// TIA Portal V17 export
// export: Created 2025-03-10T12:18:45.1065076Z, ExportSetting WithDefaults, DisplayName Totally Integrated Automation Portal, DisplayVersion V17 Update 8, DisplayName TIA Portal Openness, DisplayVersion V17 Update 8, DisplayName TIA Portal Version Control Interface, DisplayVersion V17, DisplayName SINAMICS Startdrive Advanced, DisplayVersion V17 SP2, DisplayName SINAMICS Startdrive G110M, G120, G120C, G120D, G120P, G115D, DisplayVersion V17 SP2, DisplayName SINAMICS Startdrive G130, G150, S120, S150, SINAMICS MV, S210, DisplayVersion V17 SP2, DisplayName STEP 7 Professional, DisplayVersion V17 Update 8, DisplayName SINUMERIK ONE STEP 7 Toolbox, DisplayVersion V17 Update 12, DisplayName SINUMERIK 840D sl STEP 7 Toolbox, DisplayVersion V17 Update 12, DisplayName STEP 7 Safety, DisplayVersion V17 Update 6, DisplayName WinCC Advanced, DisplayVersion V17 Update 8
FUNCTION_BLOCK "FB21011_POWDER_FEEDER_GENERAL"   // FB21011, LAD
TITLE = FB21011 POWDER FEEDER GENERAL
{ S7_Optimized_Access := 'TRUE' }
VERSION : 0.1
// stored: AutoNumber false, IsIECCheckEnabled false, IsRetainMemResEnabled false, MemoryReserve 100, SetENOAutomatically false, UDAEnableTagReadback false
   VAR_INPUT
      iPOWDER_FEEDER_BRAKER_FAULT : Bool;
      iOPERATION_MODE_LINE_1 : Word;
      iOPERATION_MODE_LINE_2 : Word;
      iOPERATION_MODE_MATCHED_LINE_1 : Bool;
      iOPERATION_MODE_MATCHED_LINE_2 : Bool;
      iFEEDER_STATE_LINE_1 : Word;
      iFEEDER_STATE_LINE_2 : Word;
      iCARRIERGAS_STATUS_LINE_1 : Bool;
      iCARRIERGAS_STATUS_LINE_2 : Bool;
      iENABLED : Bool;
   END_VAR
   VAR_OUTPUT
      oCONNECT_POWDER_FEEDER : Bool;
      oOPERATION_MODE : Word;
      oPRODUCTION_MODE : Word;
      oSYSTEM_MODE : Word;
      oSTATION_IS_ALARMS : Bool;
      oSwitchoncondition_on : Bool;
      oSwitchoncondition_off : Bool;
      oMotion_Active_Right : Bool;
      oMotion_Active_Left : Bool;
      oLimit_right : Bool;
      oLimit_left : Bool;
      oALARM_MISMATCH_FAULT : Bool;
      oALARM_FEEDER_PROFINET_MODE_FAULT : Bool;
   END_VAR
   VAR
      DATA : "POWDER FEEDER GENERAL";
      INPUT_SETTINGS : Struct
         UNIT_NUMBER : Int;
         FEEDER_NUMBER : Int;
      END_STRUCT;
   END_VAR
   VAR_TEMP
      OPTIONS_OFF : Bool;
      OPTIONS_ON : Bool;
      HOPPER_1 : Bool;
      HOPPER_2 : Bool;
      DB_NUMBER : DInt;
   END_VAR
   VAR_TEMP   // added for the SCL form of the ladder/FBD networks
      _w1 : Bool;
   END_VAR
BEGIN

NETWORK
TITLE = READ INSTANCE DB NUMBER
      L     DINO;
      +     10#800000;
      T     #DB_NUMBER;

REGION Network 2: OPTIONS OFF / Options Off
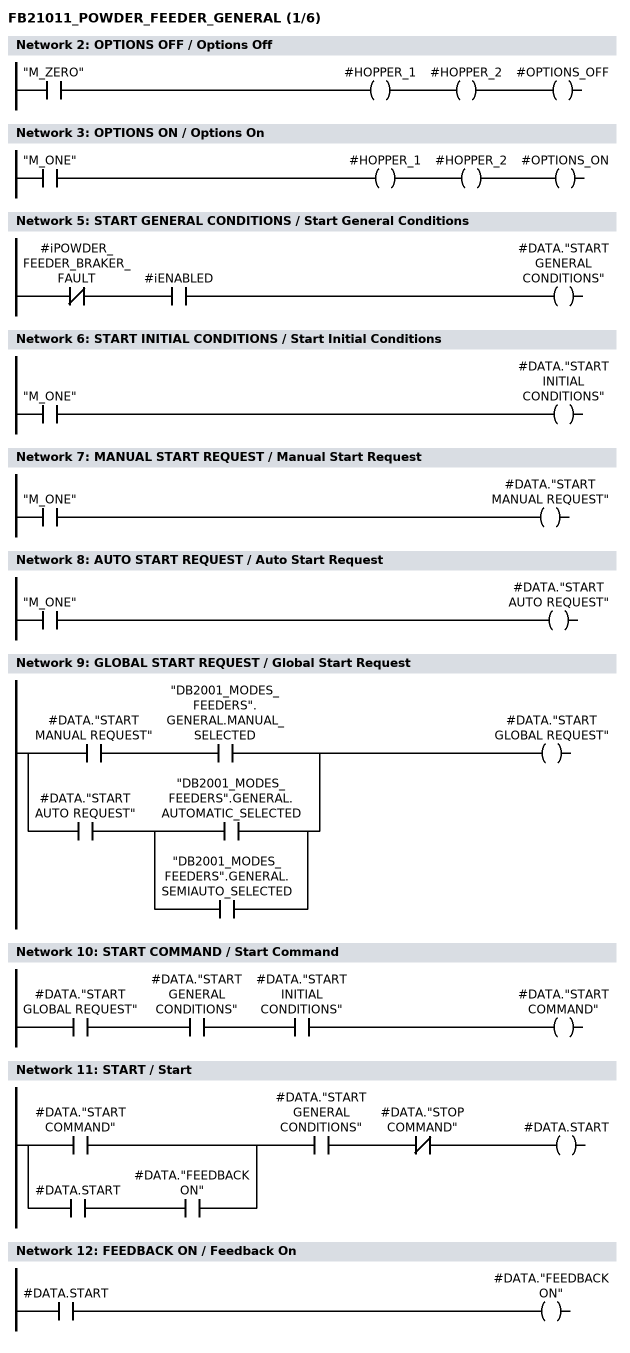
   RUNG wire#powerrail
      Contact( "M_ZERO" )
      Coil( #HOPPER_1 )
      Coil( #HOPPER_2 )
      Coil( #OPTIONS_OFF )
   END_RUNG
   // the same network as SCL:
   #HOPPER_1 := "M_ZERO";
   #HOPPER_2 := "M_ZERO";
   #OPTIONS_OFF := "M_ZERO";
END_REGION

REGION Network 3: OPTIONS ON / Options On
   RUNG wire#powerrail
      Contact( "M_ONE" )
      Coil( #HOPPER_1 )
      Coil( #HOPPER_2 )
      Coil( #OPTIONS_ON )
   END_RUNG
   // the same network as SCL:
   #HOPPER_1 := "M_ONE";
   #HOPPER_2 := "M_ONE";
   #OPTIONS_ON := "M_ONE";
END_REGION

REGION Network 4: INPUT / Input
END_REGION

REGION Network 5: START GENERAL CONDITIONS / Start General Conditions
   RUNG wire#powerrail
      I_Contact( #iPOWDER_FEEDER_BRAKER_FAULT )
      Contact( #iENABLED )
      Coil( #DATA."START GENERAL CONDITIONS" )
   END_RUNG
   // the same network as SCL:
   #DATA."START GENERAL CONDITIONS" := NOT #iPOWDER_FEEDER_BRAKER_FAULT AND #iENABLED;
END_REGION

REGION Network 6: START INITIAL CONDITIONS / Start Initial Conditions
   RUNG wire#powerrail
      Contact( "M_ONE" )
      Coil( #DATA."START INITIAL CONDITIONS" )
   END_RUNG
   // the same network as SCL:
   #DATA."START INITIAL CONDITIONS" := "M_ONE";
END_REGION

REGION Network 7: MANUAL START REQUEST / Manual Start Request
   RUNG wire#powerrail
      Contact( "M_ONE" )
      Coil( #DATA."START MANUAL REQUEST" )
   END_RUNG
   // the same network as SCL:
   #DATA."START MANUAL REQUEST" := "M_ONE";
END_REGION

REGION Network 8: AUTO START REQUEST / Auto Start Request
   RUNG wire#powerrail
      Contact( "M_ONE" )
      Coil( #DATA."START AUTO REQUEST" )
   END_RUNG
   // the same network as SCL:
   #DATA."START AUTO REQUEST" := "M_ONE";
END_REGION

REGION Network 9: GLOBAL START REQUEST / Global Start Request
   RUNG wire#powerrail
      Contact( #DATA."START MANUAL REQUEST" )
      Contact( "DB2001_MODES_FEEDERS".GENERAL.MANUAL_SELECTED )
      wire#w1
      Coil( #DATA."START GLOBAL REQUEST" )
   END_RUNG
   RUNG wire#powerrail
      Contact( #DATA."START AUTO REQUEST" )
      wire#w2
      Contact( "DB2001_MODES_FEEDERS".GENERAL.AUTOMATIC_SELECTED )
   END_RUNG wire#w1
   RUNG wire#w2
      Contact( "DB2001_MODES_FEEDERS".GENERAL.SEMIAUTO_SELECTED )
   END_RUNG wire#w1
   // the same network as SCL:
   #DATA."START GLOBAL REQUEST" := (#DATA."START MANUAL REQUEST" AND "DB2001_MODES_FEEDERS".GENERAL.MANUAL_SELECTED) OR (#DATA."START AUTO REQUEST" AND ("DB2001_MODES_FEEDERS".GENERAL.AUTOMATIC_SELECTED OR "DB2001_MODES_FEEDERS".GENERAL.SEMIAUTO_SELECTED));
END_REGION

REGION Network 10: START COMMAND / Start Command
   RUNG wire#powerrail
      Contact( #DATA."START GLOBAL REQUEST" )
      Contact( #DATA."START GENERAL CONDITIONS" )
      Contact( #DATA."START INITIAL CONDITIONS" )
      Coil( #DATA."START COMMAND" )
   END_RUNG
   // the same network as SCL:
   #DATA."START COMMAND" := #DATA."START GLOBAL REQUEST" AND #DATA."START GENERAL CONDITIONS" AND #DATA."START INITIAL CONDITIONS";
END_REGION

REGION Network 11: START / Start
   RUNG wire#powerrail
      Contact( #DATA."START COMMAND" )
      wire#w1
      Contact( #DATA."START GENERAL CONDITIONS" )
      I_Contact( #DATA."STOP COMMAND" )
      Coil( #DATA.START )
   END_RUNG
   RUNG wire#powerrail
      Contact( #DATA.START )
      Contact( #DATA."FEEDBACK ON" )
   END_RUNG wire#w1
   // the same network as SCL:
   #DATA.START := (#DATA."START COMMAND" OR (#DATA.START AND #DATA."FEEDBACK ON")) AND #DATA."START GENERAL CONDITIONS" AND NOT #DATA."STOP COMMAND";
END_REGION

REGION Network 12: FEEDBACK ON / Feedback On
   RUNG wire#powerrail
      Contact( #DATA.START )
      Coil( #DATA."FEEDBACK ON" )
   END_RUNG
   // the same network as SCL:
   #DATA."FEEDBACK ON" := #DATA.START;
END_REGION

REGION Network 13: STOP GENERAL CONDITIONS / Stop General Conditions
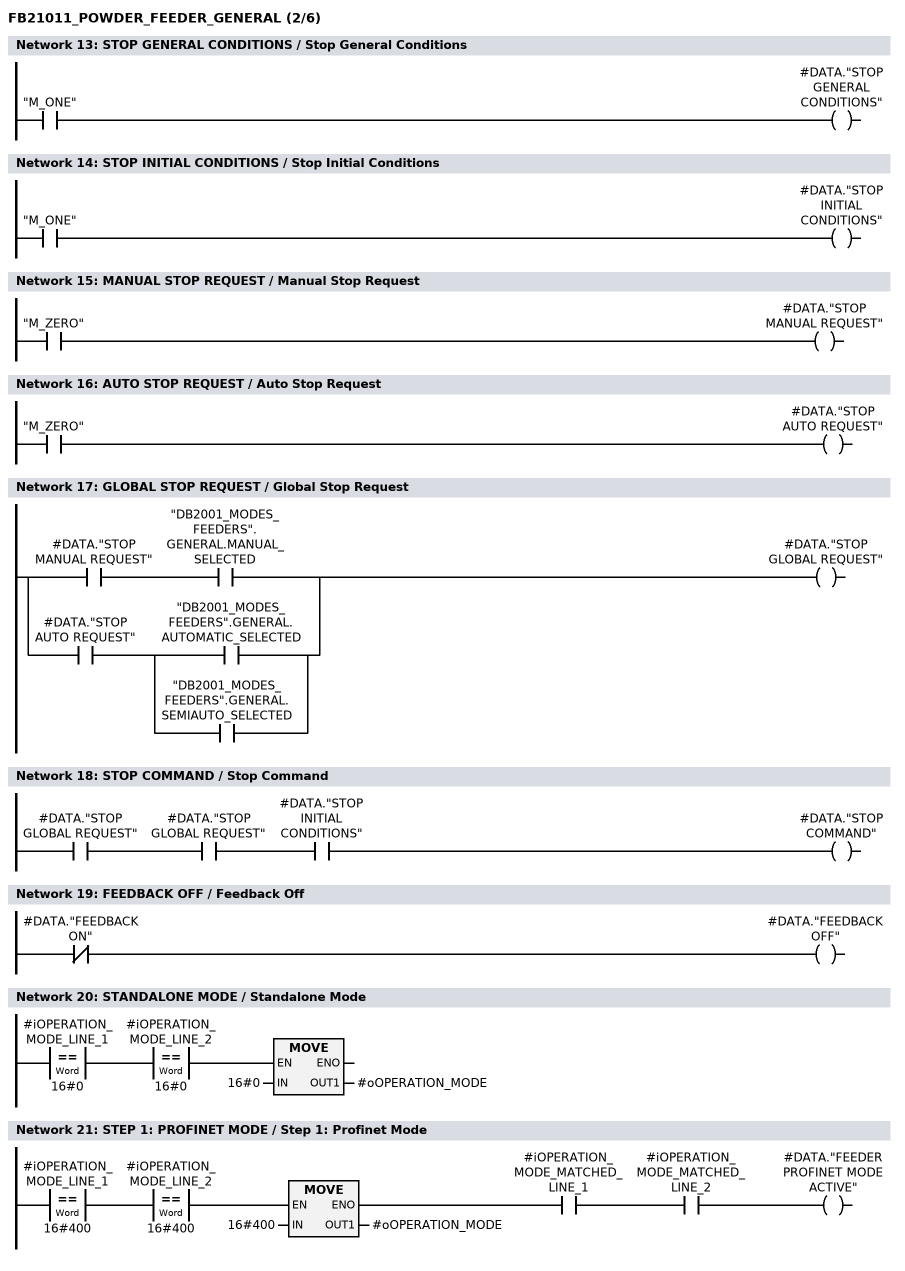
   RUNG wire#powerrail
      Contact( "M_ONE" )
      Coil( #DATA."STOP GENERAL CONDITIONS" )
   END_RUNG
   // the same network as SCL:
   #DATA."STOP GENERAL CONDITIONS" := "M_ONE";
END_REGION

REGION Network 14: STOP INITIAL CONDITIONS / Stop Initial Conditions
   RUNG wire#powerrail
      Contact( "M_ONE" )
      Coil( #DATA."STOP INITIAL CONDITIONS" )
   END_RUNG
   // the same network as SCL:
   #DATA."STOP INITIAL CONDITIONS" := "M_ONE";
END_REGION

REGION Network 15: MANUAL STOP REQUEST / Manual Stop Request
   RUNG wire#powerrail
      Contact( "M_ZERO" )
      Coil( #DATA."STOP MANUAL REQUEST" )
   END_RUNG
   // the same network as SCL:
   #DATA."STOP MANUAL REQUEST" := "M_ZERO";
END_REGION

REGION Network 16: AUTO STOP REQUEST / Auto Stop Request
   RUNG wire#powerrail
      Contact( "M_ZERO" )
      Coil( #DATA."STOP AUTO REQUEST" )
   END_RUNG
   // the same network as SCL:
   #DATA."STOP AUTO REQUEST" := "M_ZERO";
END_REGION

REGION Network 17: GLOBAL STOP REQUEST / Global Stop Request
   RUNG wire#powerrail
      Contact( #DATA."STOP MANUAL REQUEST" )
      Contact( "DB2001_MODES_FEEDERS".GENERAL.MANUAL_SELECTED )
      wire#w1
      Coil( #DATA."STOP GLOBAL REQUEST" )
   END_RUNG
   RUNG wire#powerrail
      Contact( #DATA."STOP AUTO REQUEST" )
      wire#w2
      Contact( "DB2001_MODES_FEEDERS".GENERAL.AUTOMATIC_SELECTED )
   END_RUNG wire#w1
   RUNG wire#w2
      Contact( "DB2001_MODES_FEEDERS".GENERAL.SEMIAUTO_SELECTED )
   END_RUNG wire#w1
   // the same network as SCL:
   #DATA."STOP GLOBAL REQUEST" := (#DATA."STOP MANUAL REQUEST" AND "DB2001_MODES_FEEDERS".GENERAL.MANUAL_SELECTED) OR (#DATA."STOP AUTO REQUEST" AND ("DB2001_MODES_FEEDERS".GENERAL.AUTOMATIC_SELECTED OR "DB2001_MODES_FEEDERS".GENERAL.SEMIAUTO_SELECTED));
END_REGION

REGION Network 18: STOP COMMAND / Stop Command
   RUNG wire#powerrail
      Contact( #DATA."STOP GLOBAL REQUEST" )
      Contact( #DATA."STOP GLOBAL REQUEST" )
      Contact( #DATA."STOP INITIAL CONDITIONS" )
      Coil( #DATA."STOP COMMAND" )
   END_RUNG
   // the same network as SCL:
   #DATA."STOP COMMAND" := #DATA."STOP GLOBAL REQUEST" AND #DATA."STOP GLOBAL REQUEST" AND #DATA."STOP INITIAL CONDITIONS";
END_REGION

REGION Network 19: FEEDBACK OFF / Feedback Off
   RUNG wire#powerrail
      I_Contact( #DATA."FEEDBACK ON" )
      Coil( #DATA."FEEDBACK OFF" )
   END_RUNG
   // the same network as SCL:
   #DATA."FEEDBACK OFF" := NOT #DATA."FEEDBACK ON";
END_REGION

REGION Network 20: STANDALONE MODE / Standalone Mode
   RUNG wire#powerrail
      { S7_Templates := "SrcType := Word" } EQ_Contact(in1 := #iOPERATION_MODE_LINE_1, in2 := 16#0)
      { S7_Templates := "SrcType := Word" } EQ_Contact(in1 := #iOPERATION_MODE_LINE_2, in2 := 16#0)
      Move(in := 16#0, out1 => #oOPERATION_MODE)
   END_RUNG
   // the same network as SCL:
   IF (#iOPERATION_MODE_LINE_1 = 16#0) AND (#iOPERATION_MODE_LINE_2 = 16#0) THEN
       #oOPERATION_MODE := 16#0;
   END_IF;
END_REGION

REGION Network 21: STEP 1: PROFINET MODE / Step 1: Profinet Mode
   RUNG wire#powerrail
      { S7_Templates := "SrcType := Word" } EQ_Contact(in1 := #iOPERATION_MODE_LINE_1, in2 := 16#400)
      { S7_Templates := "SrcType := Word" } EQ_Contact(in1 := #iOPERATION_MODE_LINE_2, in2 := 16#400)
      Move(in := 16#400, out1 => #oOPERATION_MODE)
      Contact( #iOPERATION_MODE_MATCHED_LINE_1 )
      Contact( #iOPERATION_MODE_MATCHED_LINE_2 )
      Coil( #DATA."FEEDER PROFINET MODE ACTIVE" )
   END_RUNG
   // the same network as SCL:
   #_w1 := (#iOPERATION_MODE_LINE_1 = 16#400) AND (#iOPERATION_MODE_LINE_2 = 16#400);
   IF #_w1 THEN #oOPERATION_MODE := 16#400; END_IF;
   #DATA."FEEDER PROFINET MODE ACTIVE" := #_w1 AND #iOPERATION_MODE_MATCHED_LINE_1 AND #iOPERATION_MODE_MATCHED_LINE_2;
END_REGION

REGION Network 22: STEP 2: PRODUCTION MODE / Step 2: Production Mode
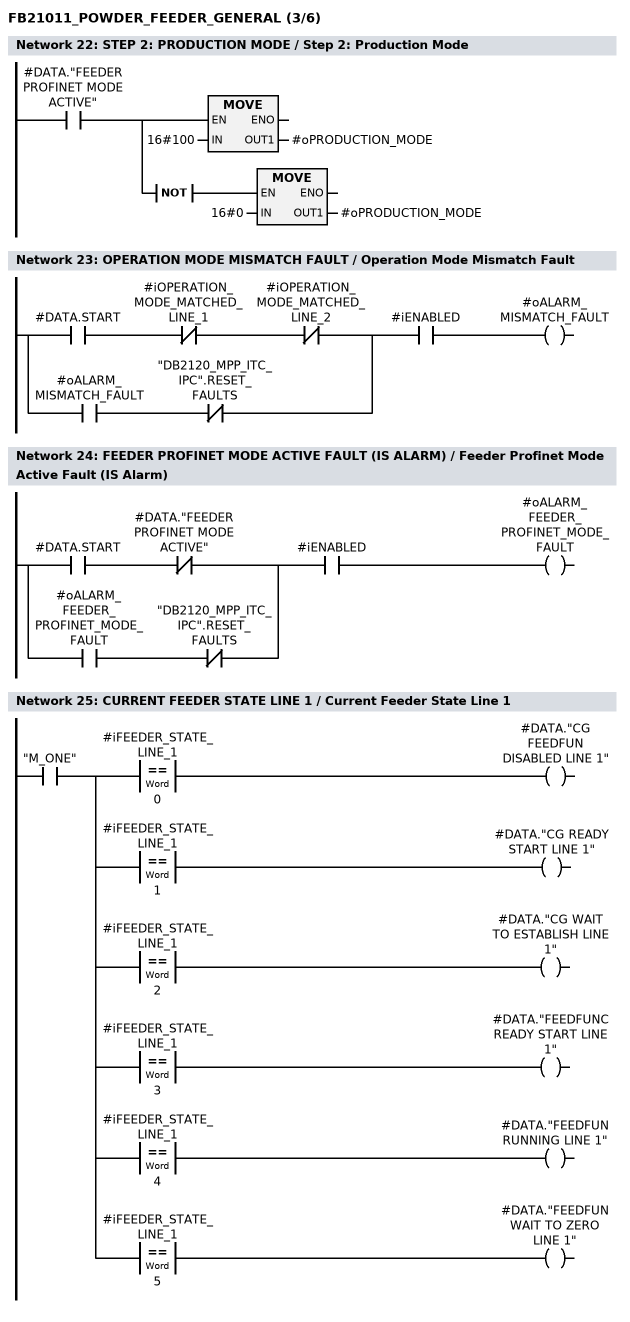
   RUNG wire#powerrail
      Contact( #DATA."FEEDER PROFINET MODE ACTIVE" )
      wire#w1
      Move(in := 16#100, out1 => #oPRODUCTION_MODE)
   END_RUNG
   RUNG wire#w1
      Not()
      Move(in := 16#0, out1 => #oPRODUCTION_MODE)
   END_RUNG
   // the same network as SCL:
   IF #DATA."FEEDER PROFINET MODE ACTIVE" THEN #oPRODUCTION_MODE := 16#100; END_IF;
   IF NOT #DATA."FEEDER PROFINET MODE ACTIVE" THEN #oPRODUCTION_MODE := 16#0; END_IF;
END_REGION

REGION Network 23: OPERATION MODE MISMATCH FAULT / Operation Mode Mismatch Fault
   RUNG wire#powerrail
      Contact( #DATA.START )
      I_Contact( #iOPERATION_MODE_MATCHED_LINE_1 )
      I_Contact( #iOPERATION_MODE_MATCHED_LINE_2 )
      wire#w1
      Contact( #iENABLED )
      Coil( #oALARM_MISMATCH_FAULT )
   END_RUNG
   RUNG wire#powerrail
      Contact( #oALARM_MISMATCH_FAULT )
      I_Contact( "DB2120_MPP_ITC_IPC".RESET_FAULTS )
   END_RUNG wire#w1
   // the same network as SCL:
   #oALARM_MISMATCH_FAULT := ((#DATA.START AND NOT #iOPERATION_MODE_MATCHED_LINE_1 AND NOT #iOPERATION_MODE_MATCHED_LINE_2) OR (#oALARM_MISMATCH_FAULT AND NOT "DB2120_MPP_ITC_IPC".RESET_FAULTS)) AND #iENABLED;
END_REGION

REGION Network 24: FEEDER PROFINET MODE ACTIVE FAULT (IS ALARM) / Feeder Profinet Mode Active Fault (IS Alarm)
   RUNG wire#powerrail
      Contact( #DATA.START )
      I_Contact( #DATA."FEEDER PROFINET MODE ACTIVE" )
      wire#w1
      Contact( #iENABLED )
      Coil( #oALARM_FEEDER_PROFINET_MODE_FAULT )
   END_RUNG
   RUNG wire#powerrail
      Contact( #oALARM_FEEDER_PROFINET_MODE_FAULT )
      I_Contact( "DB2120_MPP_ITC_IPC".RESET_FAULTS )
   END_RUNG wire#w1
   // the same network as SCL:
   #oALARM_FEEDER_PROFINET_MODE_FAULT := ((#DATA.START AND NOT #DATA."FEEDER PROFINET MODE ACTIVE") OR (#oALARM_FEEDER_PROFINET_MODE_FAULT AND NOT "DB2120_MPP_ITC_IPC".RESET_FAULTS)) AND #iENABLED;
END_REGION

REGION Network 25: CURRENT FEEDER STATE LINE 1 / Current Feeder State Line 1
   RUNG wire#powerrail
      Contact( "M_ONE" )
      wire#w1
      { S7_Templates := "SrcType := Word" } EQ_Contact(in1 := #iFEEDER_STATE_LINE_1, in2 := 0)
      Coil( #DATA."CG FEEDFUN DISABLED LINE 1" )
   END_RUNG
   RUNG wire#w1
      { S7_Templates := "SrcType := Word" } EQ_Contact(in1 := #iFEEDER_STATE_LINE_1, in2 := 1)
      Coil( #DATA."CG READY START LINE 1" )
   END_RUNG
   RUNG wire#w1
      { S7_Templates := "SrcType := Word" } EQ_Contact(in1 := #iFEEDER_STATE_LINE_1, in2 := 2)
      Coil( #DATA."CG WAIT TO ESTABLISH LINE 1" )
   END_RUNG
   RUNG wire#w1
      { S7_Templates := "SrcType := Word" } EQ_Contact(in1 := #iFEEDER_STATE_LINE_1, in2 := 3)
      Coil( #DATA."FEEDFUNC READY START LINE 1" )
   END_RUNG
   RUNG wire#w1
      { S7_Templates := "SrcType := Word" } EQ_Contact(in1 := #iFEEDER_STATE_LINE_1, in2 := 4)
      Coil( #DATA."FEEDFUN RUNNING LINE 1" )
   END_RUNG
   RUNG wire#w1
      { S7_Templates := "SrcType := Word" } EQ_Contact(in1 := #iFEEDER_STATE_LINE_1, in2 := 5)
      Coil( #DATA."FEEDFUN WAIT TO ZERO LINE 1" )
   END_RUNG
   // the same network as SCL:
   #DATA."CG FEEDFUN DISABLED LINE 1" := "M_ONE" AND (#iFEEDER_STATE_LINE_1 = 0);
   #DATA."CG READY START LINE 1" := "M_ONE" AND (#iFEEDER_STATE_LINE_1 = 1);
   #DATA."CG WAIT TO ESTABLISH LINE 1" := "M_ONE" AND (#iFEEDER_STATE_LINE_1 = 2);
   #DATA."FEEDFUNC READY START LINE 1" := "M_ONE" AND (#iFEEDER_STATE_LINE_1 = 3);
   #DATA."FEEDFUN RUNNING LINE 1" := "M_ONE" AND (#iFEEDER_STATE_LINE_1 = 4);
   #DATA."FEEDFUN WAIT TO ZERO LINE 1" := "M_ONE" AND (#iFEEDER_STATE_LINE_1 = 5);
END_REGION

REGION Network 26: CURRENT FEEDER STATE LINE 2 / Current Feeder State Line 2
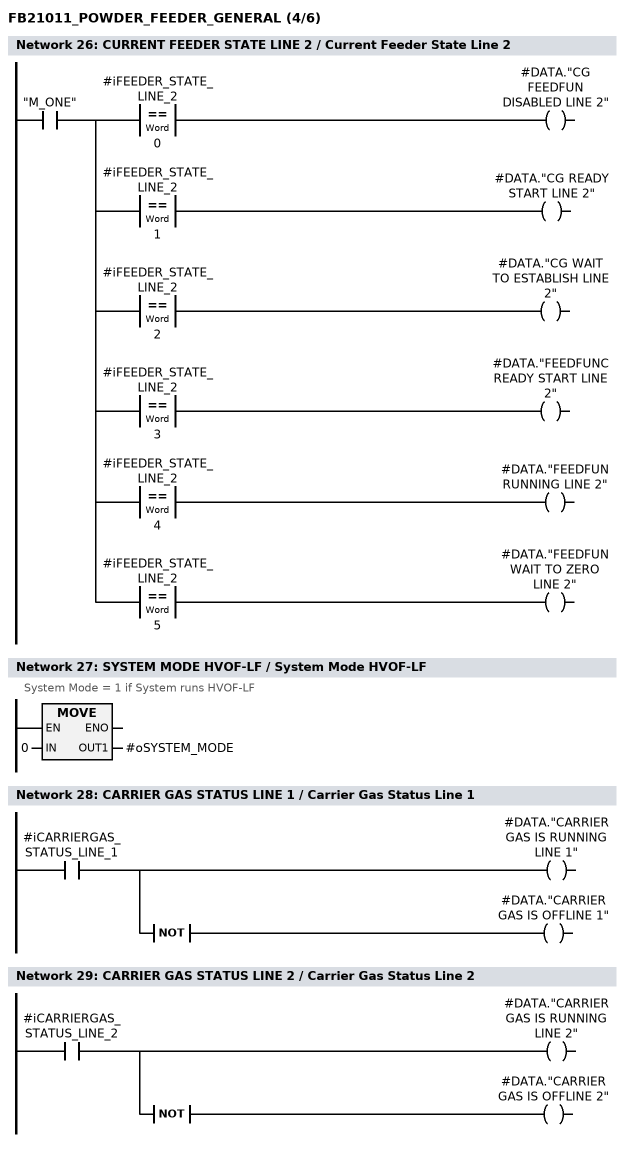
   RUNG wire#powerrail
      Contact( "M_ONE" )
      wire#w1
      { S7_Templates := "SrcType := Word" } EQ_Contact(in1 := #iFEEDER_STATE_LINE_2, in2 := 0)
      Coil( #DATA."CG FEEDFUN DISABLED LINE 2" )
   END_RUNG
   RUNG wire#w1
      { S7_Templates := "SrcType := Word" } EQ_Contact(in1 := #iFEEDER_STATE_LINE_2, in2 := 1)
      Coil( #DATA."CG READY START LINE 2" )
   END_RUNG
   RUNG wire#w1
      { S7_Templates := "SrcType := Word" } EQ_Contact(in1 := #iFEEDER_STATE_LINE_2, in2 := 2)
      Coil( #DATA."CG WAIT TO ESTABLISH LINE 2" )
   END_RUNG
   RUNG wire#w1
      { S7_Templates := "SrcType := Word" } EQ_Contact(in1 := #iFEEDER_STATE_LINE_2, in2 := 3)
      Coil( #DATA."FEEDFUNC READY START LINE 2" )
   END_RUNG
   RUNG wire#w1
      { S7_Templates := "SrcType := Word" } EQ_Contact(in1 := #iFEEDER_STATE_LINE_2, in2 := 4)
      Coil( #DATA."FEEDFUN RUNNING LINE 2" )
   END_RUNG
   RUNG wire#w1
      { S7_Templates := "SrcType := Word" } EQ_Contact(in1 := #iFEEDER_STATE_LINE_2, in2 := 5)
      Coil( #DATA."FEEDFUN WAIT TO ZERO LINE 2" )
   END_RUNG
   // the same network as SCL:
   #DATA."CG FEEDFUN DISABLED LINE 2" := "M_ONE" AND (#iFEEDER_STATE_LINE_2 = 0);
   #DATA."CG READY START LINE 2" := "M_ONE" AND (#iFEEDER_STATE_LINE_2 = 1);
   #DATA."CG WAIT TO ESTABLISH LINE 2" := "M_ONE" AND (#iFEEDER_STATE_LINE_2 = 2);
   #DATA."FEEDFUNC READY START LINE 2" := "M_ONE" AND (#iFEEDER_STATE_LINE_2 = 3);
   #DATA."FEEDFUN RUNNING LINE 2" := "M_ONE" AND (#iFEEDER_STATE_LINE_2 = 4);
   #DATA."FEEDFUN WAIT TO ZERO LINE 2" := "M_ONE" AND (#iFEEDER_STATE_LINE_2 = 5);
END_REGION

REGION Network 27: SYSTEM MODE HVOF-LF / System Mode HVOF-LF
   // System Mode = 1 if System runs HVOF-LF
   RUNG wire#powerrail
      Move(in := 0, out1 => #oSYSTEM_MODE)
   END_RUNG
   // the same network as SCL:
   #oSYSTEM_MODE := 0;
END_REGION

REGION Network 28: CARRIER GAS STATUS LINE 1 / Carrier Gas Status Line 1
   RUNG wire#powerrail
      Contact( #iCARRIERGAS_STATUS_LINE_1 )
      wire#w1
      Coil( #DATA."CARRIER GAS IS RUNNING LINE 1" )
   END_RUNG
   RUNG wire#w1
      Not()
      Coil( #DATA."CARRIER GAS IS OFFLINE 1" )
   END_RUNG
   // the same network as SCL:
   #DATA."CARRIER GAS IS RUNNING LINE 1" := #iCARRIERGAS_STATUS_LINE_1;
   #DATA."CARRIER GAS IS OFFLINE 1" := NOT #iCARRIERGAS_STATUS_LINE_1;
END_REGION

REGION Network 29: CARRIER GAS STATUS LINE 2 / Carrier Gas Status Line 2
   RUNG wire#powerrail
      Contact( #iCARRIERGAS_STATUS_LINE_2 )
      wire#w1
      Coil( #DATA."CARRIER GAS IS RUNNING LINE 2" )
   END_RUNG
   RUNG wire#w1
      Not()
      Coil( #DATA."CARRIER GAS IS OFFLINE 2" )
   END_RUNG
   // the same network as SCL:
   #DATA."CARRIER GAS IS RUNNING LINE 2" := #iCARRIERGAS_STATUS_LINE_2;
   #DATA."CARRIER GAS IS OFFLINE 2" := NOT #iCARRIERGAS_STATUS_LINE_2;
END_REGION

REGION Network 30: INMEDIATE STOP ALARMS / Inmediate Stop Alarms
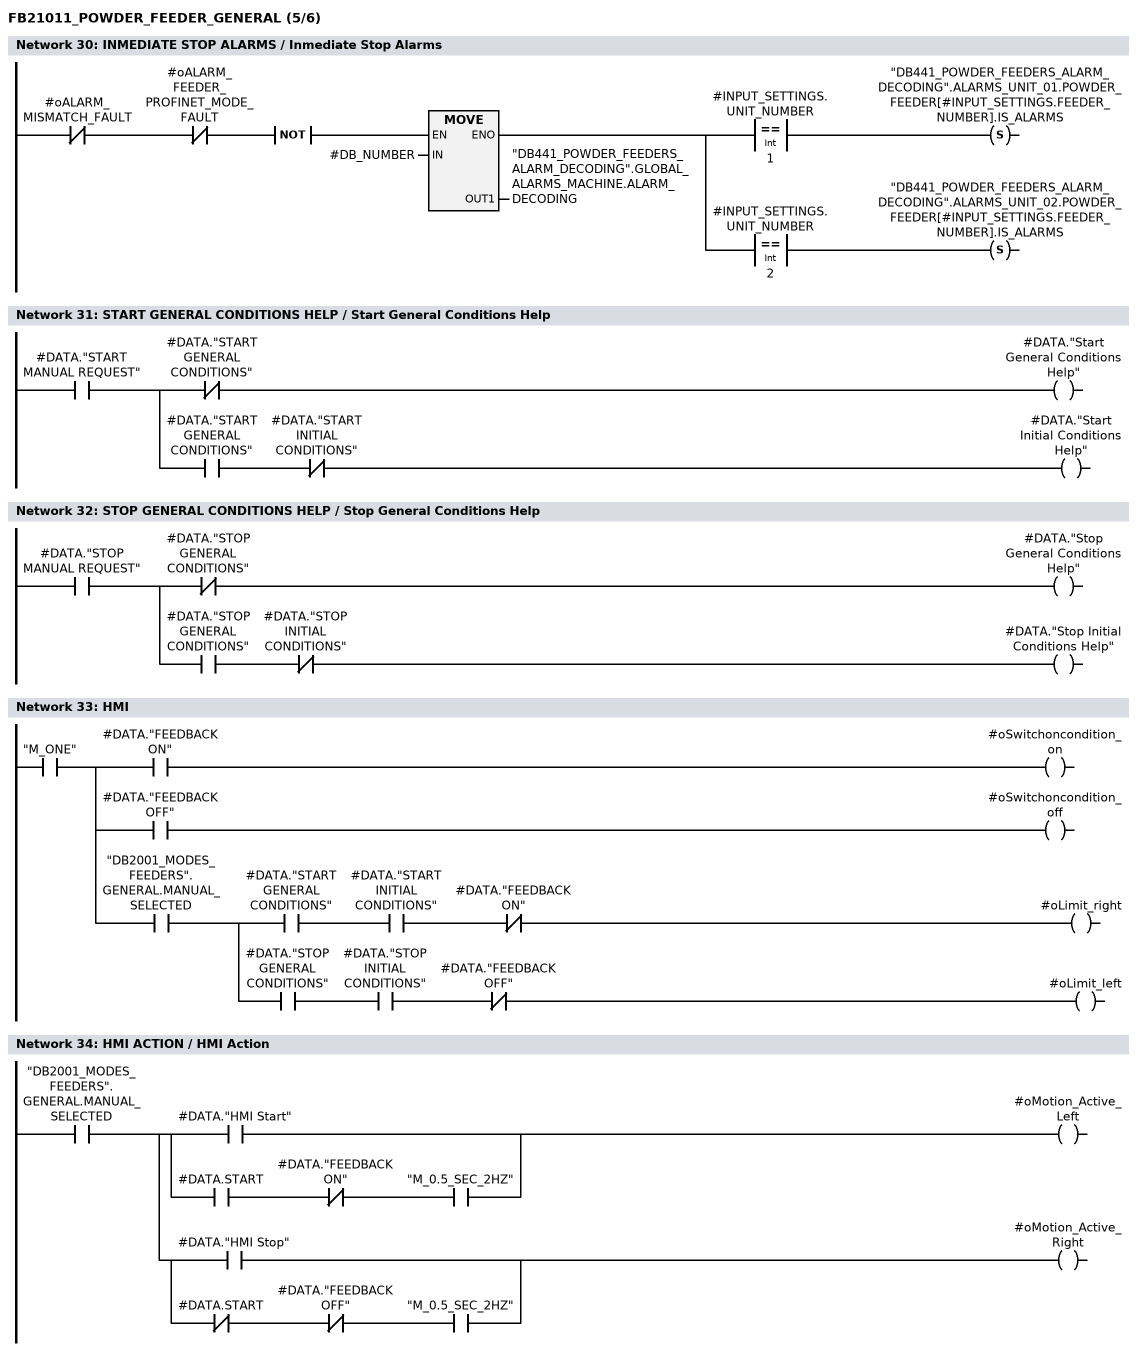
   RUNG wire#powerrail
      I_Contact( #oALARM_MISMATCH_FAULT )
      I_Contact( #oALARM_FEEDER_PROFINET_MODE_FAULT )
      Not()
      Move(in := #DB_NUMBER, out1 => "DB441_POWDER_FEEDERS_ALARM_DECODING".GLOBAL_ALARMS_MACHINE.ALARM_DECODING)
      wire#w1
      { S7_Templates := "SrcType := Int" } EQ_Contact(in1 := #INPUT_SETTINGS.UNIT_NUMBER, in2 := 1)
      S_Coil( "DB441_POWDER_FEEDERS_ALARM_DECODING".ALARMS_UNIT_01.POWDER_FEEDER[#INPUT_SETTINGS.FEEDER_NUMBER].IS_ALARMS )
   END_RUNG
   RUNG wire#w1
      { S7_Templates := "SrcType := Int" } EQ_Contact(in1 := #INPUT_SETTINGS.UNIT_NUMBER, in2 := 2)
      S_Coil( "DB441_POWDER_FEEDERS_ALARM_DECODING".ALARMS_UNIT_02.POWDER_FEEDER[#INPUT_SETTINGS.FEEDER_NUMBER].IS_ALARMS )
   END_RUNG
   // the same network as SCL:
   #_w1 := NOT (NOT #oALARM_MISMATCH_FAULT AND NOT #oALARM_FEEDER_PROFINET_MODE_FAULT);
   IF #_w1 THEN
       "DB441_POWDER_FEEDERS_ALARM_DECODING".GLOBAL_ALARMS_MACHINE.ALARM_DECODING := #DB_NUMBER;
   END_IF;
   IF #_w1 AND (#INPUT_SETTINGS.UNIT_NUMBER = 1) THEN
       "DB441_POWDER_FEEDERS_ALARM_DECODING".ALARMS_UNIT_01.POWDER_FEEDER[#INPUT_SETTINGS.FEEDER_NUMBER].IS_ALARMS := TRUE;
   END_IF;
   IF #_w1 AND (#INPUT_SETTINGS.UNIT_NUMBER = 2) THEN
       "DB441_POWDER_FEEDERS_ALARM_DECODING".ALARMS_UNIT_02.POWDER_FEEDER[#INPUT_SETTINGS.FEEDER_NUMBER].IS_ALARMS := TRUE;
   END_IF;
END_REGION

REGION Network 31: START GENERAL CONDITIONS HELP / Start General Conditions Help
   RUNG wire#powerrail
      Contact( #DATA."START MANUAL REQUEST" )
      wire#w1
      I_Contact( #DATA."START GENERAL CONDITIONS" )
      Coil( #DATA."Start General Conditions Help" )
   END_RUNG
   RUNG wire#w1
      Contact( #DATA."START GENERAL CONDITIONS" )
      I_Contact( #DATA."START INITIAL CONDITIONS" )
      Coil( #DATA."Start Initial Conditions Help" )
   END_RUNG
   // the same network as SCL:
   #DATA."Start General Conditions Help" := #DATA."START MANUAL REQUEST" AND NOT #DATA."START GENERAL CONDITIONS";
   #DATA."Start Initial Conditions Help" := #DATA."START MANUAL REQUEST" AND #DATA."START GENERAL CONDITIONS" AND NOT #DATA."START INITIAL CONDITIONS";
END_REGION

REGION Network 32: STOP GENERAL CONDITIONS HELP / Stop General Conditions Help
   RUNG wire#powerrail
      Contact( #DATA."STOP MANUAL REQUEST" )
      wire#w1
      I_Contact( #DATA."STOP GENERAL CONDITIONS" )
      Coil( #DATA."Stop General Conditions Help" )
   END_RUNG
   RUNG wire#w1
      Contact( #DATA."STOP GENERAL CONDITIONS" )
      I_Contact( #DATA."STOP INITIAL CONDITIONS" )
      Coil( #DATA."Stop Initial Conditions Help" )
   END_RUNG
   // the same network as SCL:
   #DATA."Stop General Conditions Help" := #DATA."STOP MANUAL REQUEST" AND NOT #DATA."STOP GENERAL CONDITIONS";
   #DATA."Stop Initial Conditions Help" := #DATA."STOP MANUAL REQUEST" AND #DATA."STOP GENERAL CONDITIONS" AND NOT #DATA."STOP INITIAL CONDITIONS";
END_REGION

REGION Network 33: HMI
   RUNG wire#powerrail
      Contact( "M_ONE" )
      wire#w1
      Contact( #DATA."FEEDBACK ON" )
      Coil( #oSwitchoncondition_on )
   END_RUNG
   RUNG wire#w1
      Contact( #DATA."FEEDBACK OFF" )
      Coil( #oSwitchoncondition_off )
   END_RUNG
   RUNG wire#w1
      Contact( "DB2001_MODES_FEEDERS".GENERAL.MANUAL_SELECTED )
      wire#w2
      Contact( #DATA."START GENERAL CONDITIONS" )
      Contact( #DATA."START INITIAL CONDITIONS" )
      I_Contact( #DATA."FEEDBACK ON" )
      Coil( #oLimit_right )
   END_RUNG
   RUNG wire#w2
      Contact( #DATA."STOP GENERAL CONDITIONS" )
      Contact( #DATA."STOP INITIAL CONDITIONS" )
      I_Contact( #DATA."FEEDBACK OFF" )
      Coil( #oLimit_left )
   END_RUNG
   // the same network as SCL:
   #oSwitchoncondition_on := "M_ONE" AND #DATA."FEEDBACK ON";
   #oSwitchoncondition_off := "M_ONE" AND #DATA."FEEDBACK OFF";
   #_w1 := "M_ONE" AND "DB2001_MODES_FEEDERS".GENERAL.MANUAL_SELECTED;
   #oLimit_right := #_w1 AND #DATA."START GENERAL CONDITIONS" AND #DATA."START INITIAL CONDITIONS" AND NOT #DATA."FEEDBACK ON";
   #oLimit_left := #_w1 AND #DATA."STOP GENERAL CONDITIONS" AND #DATA."STOP INITIAL CONDITIONS" AND NOT #DATA."FEEDBACK OFF";
END_REGION

REGION Network 34: HMI ACTION / HMI Action
   RUNG wire#powerrail
      Contact( "DB2001_MODES_FEEDERS".GENERAL.MANUAL_SELECTED )
      wire#w1
      Contact( #DATA."HMI Start" )
      wire#w2
      Coil( #oMotion_Active_Left )
   END_RUNG
   RUNG wire#w1
      Contact( #DATA.START )
      I_Contact( #DATA."FEEDBACK ON" )
      Contact( "M_0.5_SEC_2HZ" )
   END_RUNG wire#w2
   RUNG wire#w1
      Contact( #DATA."HMI Stop" )
      wire#w3
      Coil( #oMotion_Active_Right )
   END_RUNG
   RUNG wire#w1
      I_Contact( #DATA.START )
      I_Contact( #DATA."FEEDBACK OFF" )
      Contact( "M_0.5_SEC_2HZ" )
   END_RUNG wire#w3
   // the same network as SCL:
   #oMotion_Active_Left := "DB2001_MODES_FEEDERS".GENERAL.MANUAL_SELECTED AND (#DATA."HMI Start" OR (#DATA.START AND NOT #DATA."FEEDBACK ON" AND "M_0.5_SEC_2HZ"));
   #oMotion_Active_Right := "DB2001_MODES_FEEDERS".GENERAL.MANUAL_SELECTED AND (#DATA."HMI Stop" OR (NOT #DATA.START AND NOT #DATA."FEEDBACK OFF" AND "M_0.5_SEC_2HZ"));
END_REGION

REGION Network 35: FEEDBACK ON AUX FOR HMI / Feedback On Aux for HMI
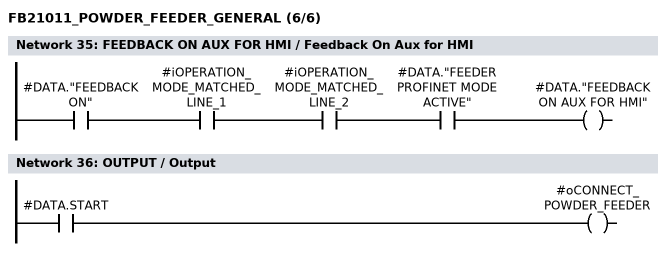
   RUNG wire#powerrail
      Contact( #DATA."FEEDBACK ON" )
      Contact( #iOPERATION_MODE_MATCHED_LINE_1 )
      Contact( #iOPERATION_MODE_MATCHED_LINE_2 )
      Contact( #DATA."FEEDER PROFINET MODE ACTIVE" )
      Coil( #DATA."FEEDBACK ON AUX FOR HMI" )
   END_RUNG
   // the same network as SCL:
   #DATA."FEEDBACK ON AUX FOR HMI" := #DATA."FEEDBACK ON" AND #iOPERATION_MODE_MATCHED_LINE_1 AND #iOPERATION_MODE_MATCHED_LINE_2 AND #DATA."FEEDER PROFINET MODE ACTIVE";
END_REGION

REGION Network 36: OUTPUT / Output
   RUNG wire#powerrail
      Contact( #DATA.START )
      Coil( #oCONNECT_POWDER_FEEDER )
   END_RUNG
   // the same network as SCL:
   #oCONNECT_POWDER_FEEDER := #DATA.START;
END_REGION
END_FUNCTION_BLOCK
